ABB RobotStudio station: EXAM.rspag

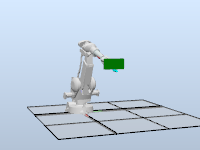
--- station ---
Station EXAM (saved by RobotStudio 20.4.9280.0)
Controller Controller60
  mechanical unit ROB_1: IRB2400_10_150__02, 6 joints, base frame (0, 0, 0) mm
Layout (positions relative to the parent item):
  - IRB2400_10_150__02 [mechanism, from Robots\IRB2400_10_150_G_02.rslib] at (0, 0, 0) mm; joint values [0.2041, 0.3579, 0.3809, 0.508, -0.4297, 1.1023] (rad or m)
  - RECTANGULARTOOL2 [part] at (1160.25, 222.53, 1120) mm, rotated rx 90 ry 0 rz 90 deg
  - Part_1 [part] at (1460.25, -777.47, 0) mm
  - Part_3 [part] at (266.55, 299.61, 2095.62) mm, rotated rx -172.42 ry 5.83 rz 0.76 deg
  - Part_4 [part]
  - Frame_1 [frame] at (1310.25, 222.53, 1000) mm
Attachment: Part_3 is attached to RECTANGULARTOOL2
Attachment: RECTANGULARTOOL2 is attached to IRB2400_10_150__02 / Link6

--- Backups/Controller60/RAPID/TASK1/PROGMOD/Module1.mod ---
MODULE Module1

    TASK PERS tooldata STATIONARY_TOOL:=[FALSE,[[1310.25,222.53,1000],[1,0,0,0]],[1,[1,1,1],[1,0,0,0],1,1,1]];
    TASK PERS wobjdata wobj1:=[TRUE,TRUE,"",[[0,0,0],[1,0,0,0]],[[0,0,0],[1,0,0,0]]];
    ! Center of Frame based in tool1 (stationary) with the orientation settled to be orizontal
    CONST robtarget CENTER_TOOL1_ORIZONTAL:=[[0, 0, 0],[0.5,-0.5,-0.5,-0.5],[0,0,-1,0],[9E+09,9E+09,9E+09,9E+09,9E+09,9E+09]];
    CONST num WALL_DISTANCE := 150;
    CONST num CYLINDER_RADIUS := 20;
    CONST num VACUUM_RADIUS := 20;
    CONST num LONG_SIDE := 400;
    CONST num SHORT_SIDE := 200;
    CONST num VacOff := VACUUM_RADIUS*0.70710678118;

    CONST robtarget HOME_POSITION:=[[873.95,222.53,1410.61],[0.5,-0.5,0.5,-0.5],[0,0,-2,0],[9E+09,9E+09,9E+09,9E+09,9E+09,9E+09]];
    CONST robtarget PSTART := [[0,-(CYLINDER_RADIUS+SHORT_SIDE/2),WALL_DISTANCE+50],[0.5,-0.5,-0.5,-0.5],[0,0,-1,0],[9E+09,9E+09,9E+09,9E+09,9E+09,9E+09]];
    CONST robtarget P0 := [[0,-(CYLINDER_RADIUS+SHORT_SIDE/2),WALL_DISTANCE],[0.5,-0.5,-0.5,-0.5],[0,0,-1,0],[9E+09,9E+09,9E+09,9E+09,9E+09,9E+09]];
    CONST robtarget P1 := [[-LONG_SIDE/2 + VACUUM_RADIUS,-(CYLINDER_RADIUS+SHORT_SIDE/2),WALL_DISTANCE],[0.5,-0.5,-0.5,-0.5],[0,0,-1,0],[9E+09,9E+09,9E+09,9E+09,9E+09,9E+09]];
    CONST robtarget P2 := [[-LONG_SIDE/2 + VACUUM_RADIUS - 2*VacOff,-(CYLINDER_RADIUS+SHORT_SIDE/2)+2*(VACUUM_RADIUS-VacOff),WALL_DISTANCE],[0.5,-0.5,-0.5,-0.5],[0,0,-1,0],[9E+09,9E+09,9E+09,9E+09,9E+09,9E+09]];
    CONST robtarget P3 := [[-LONG_SIDE/2 - VACUUM_RADIUS,-(CYLINDER_RADIUS+SHORT_SIDE/2)+2*VACUUM_RADIUS,WALL_DISTANCE],[0.5,-0.5,-0.5,-0.5],[0,0,-1,0],[9E+09,9E+09,9E+09,9E+09,9E+09,9E+09]];
    CONST robtarget P4 := [[-LONG_SIDE/2 - VACUUM_RADIUS,(CYLINDER_RADIUS+SHORT_SIDE/2)-2*VACUUM_RADIUS,WALL_DISTANCE],[0.5,-0.5,-0.5,-0.5],[0,0,-1,0],[9E+09,9E+09,9E+09,9E+09,9E+09,9E+09]];
    CONST robtarget P5 := [[-LONG_SIDE/2 + VACUUM_RADIUS - 2*VacOff,-(CYLINDER_RADIUS-SHORT_SIDE/2)+2*(VACUUM_RADIUS)-VacOff,WALL_DISTANCE],[0.5,-0.5,-0.5,-0.5],[0,0,-1,0],[9E+09,9E+09,9E+09,9E+09,9E+09,9E+09]];
    CONST robtarget P6 := [[-LONG_SIDE/2 + VACUUM_RADIUS,(CYLINDER_RADIUS+SHORT_SIDE/2),WALL_DISTANCE],[0.5,-0.5,-0.5,-0.5],[0,0,-1,0],[9E+09,9E+09,9E+09,9E+09,9E+09,9E+09]];
    CONST robtarget P7 := [[+LONG_SIDE/2 - VACUUM_RADIUS,(CYLINDER_RADIUS+SHORT_SIDE/2),WALL_DISTANCE],[0.5,-0.5,-0.5,-0.5],[0,0,-1,0],[9E+09,9E+09,9E+09,9E+09,9E+09,9E+09]];
    CONST robtarget P8 := [[+LONG_SIDE/2 - VACUUM_RADIUS + 2*VacOff,-(CYLINDER_RADIUS-SHORT_SIDE/2)+2*(VACUUM_RADIUS)-VacOff,WALL_DISTANCE],[0.5,-0.5,-0.5,-0.5],[0,0,-1,0],[9E+09,9E+09,9E+09,9E+09,9E+09,9E+09]];
    CONST robtarget P9 := [[+LONG_SIDE/2 + VACUUM_RADIUS,(CYLINDER_RADIUS+SHORT_SIDE/2)-2*VACUUM_RADIUS,WALL_DISTANCE],[0.5,-0.5,-0.5,-0.5],[0,0,-1,0],[9E+09,9E+09,9E+09,9E+09,9E+09,9E+09]];
    CONST robtarget P10 := [[+LONG_SIDE/2 + VACUUM_RADIUS,-(CYLINDER_RADIUS+SHORT_SIDE/2)+2*VACUUM_RADIUS,WALL_DISTANCE],[0.5,-0.5,-0.5,-0.5],[0,0,-1,0],[9E+09,9E+09,9E+09,9E+09,9E+09,9E+09]];
    CONST robtarget P11 := [[+LONG_SIDE/2 - VACUUM_RADIUS + 2*VacOff,-(CYLINDER_RADIUS+SHORT_SIDE/2)+2*(VACUUM_RADIUS-VacOff),WALL_DISTANCE],[0.5,-0.5,-0.5,-0.5],[0,0,-1,0],[9E+09,9E+09,9E+09,9E+09,9E+09,9E+09]];
    CONST robtarget P12 := [[+LONG_SIDE/2 - VACUUM_RADIUS,-(CYLINDER_RADIUS+SHORT_SIDE/2),WALL_DISTANCE],[0.5,-0.5,-0.5,-0.5],[0,0,-1,0],[9E+09,9E+09,9E+09,9E+09,9E+09,9E+09]];

    !***********************************************************
    !
    ! Module: Module1
    !
    ! Description:
    ! <Insert description here>
    !
    ! Author: Donato Caramia AND Giovanni Soleti
    !
    ! Version: 1.0
    !
    !***********************************************************


    !***********************************************************
    !
    ! Procedure main
    !
    ! This is the entry point of your program
    !
    !***********************************************************
    PROC main()
        !Set the robot in Home Position
        MoveL HOME_POSITION, v200, z50, tool0;

        MoveL PSTART, v200, z50, STATIONARY_TOOL\WObj:=wobj1;
        MoveL P0, v200, z50, STATIONARY_TOOL\WObj:=wobj1;
        MoveL P1, v200, z50, STATIONARY_TOOL\WObj:=wobj1;
        MoveC P2,P3, v200, z50, STATIONARY_TOOL\WObj:=wobj1;
        MoveL P4, v200, z50, STATIONARY_TOOL\WObj:=wobj1;
        MoveC P5,P6, v200, z50, STATIONARY_TOOL\WObj:=wobj1;
        MoveL P7, v200, z50, STATIONARY_TOOL\WObj:=wobj1;
        MoveC P8,P9, v200, z50, STATIONARY_TOOL\WObj:=wobj1;
        MoveL P10, v200, z50, STATIONARY_TOOL\WObj:=wobj1;
        MoveC P11,P12, v200, z50, STATIONARY_TOOL\WObj:=wobj1;
        MoveL P0, v200, z50, STATIONARY_TOOL\WObj:=wobj1;
    ENDPROC
ENDMODULE

--- Backups/Controller60/RAPID/TASK1/SYSMOD/LINKEDM.sys ---
%%%
  VERSION:1
  LANGUAGE:ENGLISH
%%%

MODULE LINKEDM (SYSMODULE)

! FOLLOWER
!     Name of electronically linked follower axis used by operator at teach pendent.
      PERS string l_f_axis_name{5}       :=  ["",  "", "", "", ""];

!     Name of the mechanical unit for follower axis.
      PERS string l_f_mecunt_n{5}  :=  ["", "", "", "", ""];

!     Linked follower axis number in the mechanical unit (first axis in mech. unit is number 1).
      PERS num l_f_axis_no{5}      :=  [0,          0,   0,  0,  0];

! MASTER
!     Name of the mechanical unit for linked master axis.
      PERS string l_m_mecunt_n{5} :=  ["", "", "", "", ""];

!     Linked master axis number in the mechanical unit (first axis in mech. unit is number 1).
!     See axis number table in documentation for different master mechanical units.
      PERS num l_m_axis_no{5}     :=  [0,  0,  0,  0,  0];

! POSITION OFFSET
!     The increase of the allowed offset position between the master and follower
!     positions, used when starting AUTO mode. As soon as the offset is decreased
!     the old configurated parameter is used.
!     Example: 3 => the configurated value of allowed offset is increased 3 times.
      PERS num offset_ratio{5}       :=  [10,  10,   10,  10,  10];

! SPEED RATIO
!     Speed_ratio used in AUTO and JOG modes [ very_slow   slow    normal    fast]
!     Value 1 = max allowed manual speed.
      CONST num speed_ratio {20}      := [0.01, 0.01, 0.01, 0.01, 0.01,
                                          0.05, 0.05, 0.05, 0.05, 0.05,
                                          0.20, 0.20, 0.20, 0.20, 0.20,
                                          1.00, 1.00, 1.00, 1.00, 1.00];

! STEP SIZE
!     Displacement position used in JOG mode for each activation of positive or
!     negative movement.                  [very_short    short   normal   long]
!     Unit degees or meter.
      CONST num displacement {20}     := [0.001, 0.001, 0.001, 0.001, 0.001,
                                          0.005, 0.005, 0.005, 0.005, 0.005,
                                          0.020, 0.020, 0.020, 0.020, 0.020,
                                          0.100, 0.100, 0.100, 0.100, 0.100];


!-------------------------------------------------------------
 PROC Linked_m ()
      Linked_m_exe ;
 ENDPROC
ENDMODULE
